(* CODESYS project tc motion control.library
   Author: Adam Garner
   Placeholder: Motion
   Title: Motion
   Version: 0.1.0.0
   Company: Ljmu

Project tree, tasks and I/O mapping:
  libraries: Tc2_MC2, * (Beckhoff Automation GmbH); Tc2_MC2_Drive, * (Beckhoff Automation GmbH); Tc2_Standard, * (Beckhoff Automation GmbH); Tc2_System, * (Beckhoff Automation GmbH); Tc2_Utilities, * (Beckhoff Automation GmbH); Tc3_EventLogger, * (Beckhoff Automation GmbH); Tc3_JsonXml, * (Beckhoff Automation GmbH); Tc3_Module, * (Beckhoff Automation GmbH)
  DUTs/
    data type e_IDXError
    data type e_MCState
    data type e_MotorReadState
    data type ST_IDXError
    data type ST_IDXErrorCode
    data type ST_MCState
  GVLs/
  POUs/
    function block FB_IDXError [ST]: FB_init, GetErrorStructure, IsError, ResetError
    function block FB_IDXReadErrorCode [ST]: ParseErrorCode
    function block FB_IDXReadErrorRegister [ST]: ParseErrorRegister
    function block FB_IDXResetError [ST]
    function block FB_Motion [ST]: Enable, Estop, FB_init, GetAxisRef, GetCurrentPosition, GetStatus, Home, MoveTo, Reset
    function block FB_MotionEventSender [ST]: COEError, EnableMotor, Homing, MotorError, MoveTo, NCReset
    function block FB_ReadErrorStringFromESI [ST]: GetErrorString, StringToUint
    program MAIN [ST]
  VISUs/
*)

// DUTs/e_IDXError
{attribute 'qualified_only'}
{attribute 'strict'}
TYPE e_IDXError :
(
	Generic_Error := 0,
	Current_Error :=1,
	Voltage_Error:=2,
	Temperature_Error:=3,
	Communication_Error := 4,
	Device_Profile_Specific := 5,
	Reserved := 6,
	Motion_Error :=7
);
END_TYPE

// DUTs/e_MCState
{attribute 'qualified_only'}
{attribute 'strict'}
TYPE e_MCState :
(
	Busy,
	Done,
	Error,
	CommandAborted,
	Active,
	Idle
);
END_TYPE

// DUTs/e_MotorReadState
// -27 as is qualified only shouldnt be flagged anyway
{attribute 'strict'}
{attribute 'qualified_only'}
TYPE e_MotorReadState :
(
Idle,
ReadingErrorArray,
{attribute 'analysis' := '-27'}
Parse,
EraseErrorArray,
Waiting,
Error,
CountingErrors,
ReadNextError

);
END_TYPE

// DUTs/ST_IDXError
TYPE ST_IDXError :
STRUCT
	GenericError:BOOL;
	CurrentError : BOOL;
	VoltageError:BOOL;
	TemperatureError:BOOL;
	Communication_Error :BOOL;
	DeviceProfileSpecific :BOOL;
	Reserved :BOOL;
	MotionError :BOOL;
	ErrorCodeArr:ARRAY [0..4] OF ST_IDXErrorCode;


END_STRUCT
END_TYPE

// DUTs/ST_IDXErrorCode
TYPE ST_IDXErrorCode :
STRUCT
	ErrorCode: UINT;
	ErrorString:STRING;
	TimeCode:DT;
END_STRUCT
END_TYPE

// DUTs/ST_MCState
TYPE ST_MCState :
STRUCT
	MCState : e_MCState;
	Done:BOOL;
	CommandAborted:BOOL;
	Status :BOOL;
	Active :BOOL;
	Busy:BOOL;
	Error:BOOL;
	ErrorID:UDINT;
	
END_STRUCT
END_TYPE

// POUs/FB_IDXError
FUNCTION_BLOCK FB_IDXError
// www.maxongroup.com/medias/sys_master/root/8837359632414/IDX-Firmware-Specification-En.pdf 	
VAR
	AxisName 				:STRING;
	ExecuteRead 			: BOOL; 
	MappedErrorCode AT%I* 	: UINT;
	stIDXError 				: ST_IDXError;
	
	fbIDXErrorEventSender 	: FB_MotionEventSender;
	MotorErrorEventSent		: BOOL;


	fbIdxReadErrorCode 		: FB_IDXReadErrorCode;
	NumOfErrorCodes			: USINT;
	ErrorCodeReadError 		: BOOL;
	ErrorCodeAdsErrorCode	: UINT;
	ErrorCodeReadBusy		: BOOL;
	
	fbIDXReadErrorRegister	: FB_IDXReadErrorRegister;
	ErrorRegisterReadError 	: BOOL;
	ErrorRegisterReadBusy	: BOOL;
	ErrorRegisterAdsErrorCode: UINT;
	eErrorRegisterReadState : e_MotorReadState;
	
	fbReadErrorStringFromESI: FB_ReadErrorStringFromESI;
	ErrorStringReadReady 	: BOOL;
	ErrorStringReadBusy 	: BOOL;
	ErrorStringReadError 	: BOOL;
	ErrorStringFound 		: BOOL;
	
	CoeErrorCodeMessageSent : BOOL;
	CoeErrorregisterMessageSent : BOOL;
	
	

	

END_VAR

VAR_INPUT
	Axis 					: AXIS_REF;
END_VAR

VAR_OUTPUT
    Busy         			: BOOL;
    Error        			: BOOL;
END_VAR

VAR CONSTANT
	MaxIndex 				: USINT := 4;
END_VAR

VAR_TEMP
	TempErrorCode 			: UINT;
	TempErrorString 		: STRING;
	Index					: USINT;
END_VAR

// read error Reg 
// check for error messages availible 

IF NOT (MappedErrorCode=0) THEN
	ExecuteRead := TRUE; // motor in error state 
	
ELSE
	ExecuteRead:= FALSE;
END_IF

fbIdxReadErrorCode(
	Axis:= Axis,
	Execute:= ExecuteRead,
	NumOfErrors=> NumOfErrorCodes,
	stErrorInOut:=stIDXError,
	ReadError=>ErrorCodeReadError,
	AdsErrId=>ErrorCodeAdsErrorCode,
	ReadBusy => ErrorCodeReadBusy);

CoeErrorCodeMessageSent := fbIDXErrorEventSender.COEError(
	AxisName := AxisName,
	Error := ErrorCodeReadError,
	AdsErrId:= ErrorCodeAdsErrorCode,
	Description:= 'ErrorCodeRead');

fbIDXReadErrorRegister(
	Axis:= Axis, 
	Execute:= ExecuteRead, 
	stErrorRegisterInOut:=stIDXError , 
	ReadError=> ErrorRegisterReadError, 
	AdsErrId=> ErrorRegisterAdsErrorCode, 
	eMotorReadState=>eErrorRegisterReadState,
	ReadBusy=> ErrorRegisterReadBusy );

CoeErrorregisterMessageSent:= fbIDXErrorEventSender.COEError(
	AxisName:= AxisName,
	Error := ErrorRegisterReadError,
	AdsErrId:= ErrorRegisterAdsErrorCode,
	Description:= 'ErrorCodeRegister');


fbReadErrorStringFromESI(
	ReadyFlag=>ErrorStringReadReady,
	Busy=>ErrorStringReadBusy,
	Error=>ErrorStringReadError);


IF (ErrorStringReadReady AND ExecuteRead ) THEN
	FOR Index:=0  TO MaxIndex BY 1 DO
		TempErrorCode:= stIDXError.ErrorCodeArr[Index].ErrorCode;
		IF NOT (TempErrorCode =0) THEN
			ErrorStringFound:= fbReadErrorStringFromESI.GetErrorString(ErrorCodeIn:= TempErrorCode,ErrorStringOut=>TempErrorString);
			stIDXError.ErrorCodeArr[Index].ErrorString:= TempErrorString;
		END_IF
	END_FOR
END_IF
	
MotorErrorEventSent:= fbIDXErrorEventSender.MotorError(stIDXError:=stIDXError,AxisName:= AxisName);

Busy := ErrorStringReadBusy OR ErrorRegisterReadBusy OR ErrorCodeReadBusy;
Error := ErrorStringReadError OR ErrorRegisterReadError OR ErrorCodeReadError;

METHOD FB_init : BOOL
VAR_INPUT
	bInitRetains : BOOL; // if TRUE, the retain variables are initialized (warm start / cold start)
	bInCopyCode : BOOL;  // if TRUE, the instance afterwards gets moved into the copy code (online change)
	AxisNameIn	:String;
END_VAR
AxisName := AxisNameIn;
END_METHOD

METHOD PUBLIC GetErrorStructure 
VAR_OUTPUT
	StIDXErrorOut : ST_IDXError;
END_VAR
StIDXErrorOut:= stIDXError;
END_METHOD

// returns true if motor is in error state 
METHOD IsError : BOOL
IsError := ExecuteRead;
END_METHOD

METHOD ResetError : BOOL
VAR_IN_OUT
	   		{attribute 'analysis' := '-27'}
	Execute			: BOOL;(*Function block execution is triggered by a rising edge at this input.*)
END_VAR

VAR_INST
	fbCoEWrite		: FB_CoEWrite;
    Data       		: UINT := 16#0080;
    ReadError          	: BOOL;
    AdsErrId       	: UINT;
    CANopenErrId   	: UINT;
END_VAR

VAR CONSTANT
	NetId          	: T_AmsNetID:= '';(*netID of PC with NC*)
   	Index          	: WORD:= 16#6040;(*CoE object index*)
   	SubIndex       	: BYTE:=16#0;(*CoE sub index*)
   	Timeout        	: TIME := DEFAULT_ADS_TIMEOUT;(*States the time before the function is cancelled.*)
  	CompleteAccess 	: BOOL:= FALSE;(*Function block reads the complete object with all sub index*)
END_VAR
IF __ISVALIDREF(Execute) THEN	
	fbCoEWrite(
    NetId          := NetId, 
    Index          := Index, 
    SubIndex       := SubIndex, 
    pSrcBuf        := ADR(Data), 
    BufLen         := USINT_TO_UDINT(SIZEOF(Data)), 
    Execute        := Execute, 
    Timeout        := Timeout, 
    CompleteAccess := CompleteAccess, 
    Axis := Axis
);

END_IF

IF (NOT fbCoEWrite.Busy) AND   __ISVALIDREF(Execute) THEN
    ReadError    := fbCoEWrite.Error;
	IF (NOT ReadError) AND Execute THEN
		ResetError:= TRUE; // reset successfully only shows for one cycle
	ELSE 
		ResetError:= FALSE;
	END_IF
	
    AdsErrId     := fbCoEWrite.AdsErrId;
    CANopenErrId :=fbCoEWrite.CANopenErrId;
    Execute      := FALSE;
	IF NOT ReadError THEN
		ResetError:= TRUE; // reset successfully
	END_IF
END_IF
END_METHOD

END_FUNCTION_BLOCK

// POUs/FB_MotionEventSender
FUNCTION_BLOCK FB_MotionEventSender
VAR
	fbTcMessage : FB_TcMessage;
END_VAR

METHOD COEError : BOOL
VAR_INPUT
    Error        	: BOOL;
    AdsErrId     	: UINT;
	Description		: STRING;
	AxisName		:STRING;
END_VAR
VAR_INST
	LastError		:BOOL;

END_VAR

VAR
	SendResult 			:HRESULT;

	
END_VAR
COEError := FALSE;
IF (NOT LastError) AND Error THEN // only enter is a current error is in place and the last cycle the error was 0 
	 {analysis -9,-46} // Unused  return values and possible use of none init interfaces 
	fbTcMessage.CreateEx(TC_EVENTS.MotionEvents.CoeError,0);
	fbTcMessage.ipArguments.Clear();
	fbTcMessage.ipArguments.AddString(AxisName);
	fbTcMessage.ipArguments.AddUInt(AdsErrId);
	fbTcMessage.ipArguments.AddString(Description);
	SendResult:= fbTcMessage.Send(0);
	{analysis 9,46}
	IF (SendResult=0) THEN
		COEError := TRUE;
	END_IF
END_IF
LastError:= Error;
END_METHOD

METHOD EnableMotor : BOOL
VAR_IN_OUT
	stAxisPowerState : ST_MCState;
END_VAR
VAR_INPUT
	AxisName :STRING;
END_VAR
VAR_INST
	stLastAxisPowerState :ST_MCState;
END_VAR
VAR
	SendResult 			:HRESULT;
	SendEvent :BOOL:= FALSE;
END_VAR
EnableMotor := FALSE;

IF __ISVALIDREF(stAxisPowerState) THEN

	IF NOT (stLastAxisPowerState.MCState = stAxisPowerState.MCState) THEN // state has changed 
	 	{analysis -9,-46} // Unused  return values and possible use of none init interfaces 
		CASE(stAxisPowerState.MCState) OF
		
		e_MCState.Active:
			fbTcMessage.CreateEx(TC_EVENTS.MotionEvents.MotorEnabled,0);
			SendEvent:= TRUE;
		
		e_MCState.Error:
			fbTcMessage.CreateEx(TC_EVENTS.MotionEvents.MotorEnableError,0);
			SendEvent:= TRUE;
		
		e_MCState.Idle:
			fbTcMessage.CreateEx(TC_EVENTS.MotionEvents.MotorDisabled,0);
			SendEvent:= TRUE;
		ELSE
			SendEvent:= FALSE;
		END_CASE
	
		IF SendEvent THEN
			fbTcMessage.ipArguments.Clear();
			fbTcMessage.ipArguments.AddString(AxisName);
			SendResult:= fbTcMessage.Send(0);
			IF (SendResult=0) THEN
				EnableMotor := TRUE;
			END_IF
		END_IF
	END_IF

	stLastAxisPowerState := stAxisPowerState;
END_IF
END_METHOD

METHOD Homing : BOOL
VAR_IN_OUT
	stAxisHomeState : ST_MCState;
END_VAR
VAR_INPUT
	AxisName :STRING;
	ErrorCodeIn :UDINT;
END_VAR
VAR_INST
	stLastAxisHomeState : ST_MCState;
END_VAR
VAR
	SendEvent : BOOL;
	SendResult : Hresult;
END_VAR
Homing := FALSE;

IF  __ISVALIDREF(stAxisHomeState) THEN
	
	IF  (NOT (stLastAxisHomeState.MCState = stAxisHomeState.MCState)) THEN
		CASE(stAxisHomeState.MCState) OF 
		{analysis -9,-46} // Unused  return values and possible use of none init interfaces 
		e_MCState.Done:
			fbTcMessage.CreateEx(TC_EVENTS.MotionEvents.HomeCompleted,0);
			fbTcMessage.ipArguments.Clear();
			fbTcMessage.ipArguments.AddString(AxisName);
			SendEvent := TRUE;
		
		e_MCState.Busy:
			fbTcMessage.CreateEx(TC_EVENTS.MotionEvents.HomeCommandReceived,0);
			fbTcMessage.ipArguments.Clear();
			fbTcMessage.ipArguments.AddString(AxisName);
			SendEvent := TRUE;
		
		e_MCState.Error:
			fbTcMessage.CreateEx(TC_EVENTS.MotionEvents.HomeError,0);
			fbTcMessage.ipArguments.Clear();
			fbTcMessage.ipArguments.AddString(AxisName);
			fbTcMessage.ipArguments.AddUDInt(ErrorCodeIn);
			SendEvent := TRUE;
			
		
		e_MCState.CommandAborted:
			fbTcMessage.CreateEx(TC_EVENTS.MotionEvents.HomeAborted,0);
			fbTcMessage.ipArguments.Clear();
			fbTcMessage.ipArguments.AddString(AxisName);
			SendEvent := TRUE;
			
		e_MCState.Idle:
			SendEvent := FALSE;
		
		ELSE
			SendEvent := FALSE;
			
		
		END_CASE
		
			IF SendEvent THEN
				SendResult:= fbTcMessage.Send(0);
			
				IF (SendResult=0) THEN
					Homing := TRUE;
				END_IF
	
			END_IF
	END_IF
	
	stLastAxisHomeState:= stAxisHomeState;

END_IF
END_METHOD

METHOD PUBLIC MotorError :BOOL
VAR_IN_OUT
	stIDXError 	:ST_IDXError;
END_VAR
VAR_INPUT
	AxisName 	:STRING;
END_VAR
VAR_INST
	stLastIDXError : ST_IDXError;
END_VAR
VAR
	Index :INT;
	ErrorCodeInHex :STRING[255];
	SendResult :HRESULT;
END_VAR
VAR CONSTANT
	MaxIndex :INT := 4 ; 
END_VAR
MotorError:= FALSE;
IF __ISVALIDREF(stIDXError) THEN
FOR Index := 0 TO MaxIndex BY 1 DO 
	IF NOT ( stIDXError.ErrorCodeArr[Index].ErrorCode =stLastIDXError.ErrorCodeArr[Index].ErrorCode) THEN
		{analysis -9,-46,-130}// Unused  return values possible use of none init interfaces ,  Implicit expanding conversion 
		fbTcMessage.CreateEx(TC_EVENTS.MotionEvents.MotorError,0);
		fbTcMessage.ipArguments.Clear();
		fbTcMessage.ipArguments.AddString(AxisName);
		ErrorCodeInHex := DWORD_TO_HEXSTR(stIDXError.ErrorCodeArr[Index].ErrorCode,4,FALSE);
		fbTcMessage.ipArguments.AddString(ErrorCodeInHex);
		fbTcMessage.ipArguments.AddString(stIDXError.ErrorCodeArr[Index].ErrorString);
		SendResult := fbTcMessage.Send(0);
		{analysis 9,46,130}
		IF (SendResult=0) THEN
			MotorError:= TRUE;
		END_IF
		stLastIDXError.ErrorCodeArr[Index]:= stIDXError.ErrorCodeArr[Index];
			
	END_IF
END_FOR
END_IF
END_METHOD

// moveTo bool is true when a event has been sent 
METHOD MoveTo : BOOL
VAR_IN_OUT
	stAxisMoveState : ST_MCState;
END_VAR
VAR_INPUT
	AxisName :STRING;
	TargetPositionIn : LREAL;
	VelocityIn : LREAL;
END_VAR
VAR_INST
	stLastAxisMoveState : ST_MCState;
END_VAR
VAR
	SendEvent : BOOL;
	SendResult : Hresult;
	
END_VAR
MoveTo:= FALSE;
	
IF __ISVALIDREF(stAxisMoveState) THEN
	
	IF  (NOT (stAxisMoveState.MCState = stLastAxisMoveState.MCState)) THEN
	
		CASE(stAxisMoveState.MCState) OF 
		{analysis -9,-46} // Unused  return values and possible use of none init interfaces 	
			e_MCState.Active:
			fbTcMessage.CreateEx(TC_EVENTS.MotionEvents.MotorMoveActive,0);
			fbTcMessage.ipArguments.Clear();
			fbTcMessage.ipArguments.AddString(AxisName);
			SendEvent := TRUE;
	
		e_MCState.Busy:
			fbTcMessage.CreateEx(TC_EVENTS.MotionEvents.MoveCommandReceived,0);
			fbTcMessage.ipArguments.Clear();
			fbTcMessage.ipArguments.AddString(AxisName);
			fbTcMessage.ipArguments.AddLReal(TargetPositionIn);
			fbTcMessage.ipArguments.AddLReal(VelocityIn);
			SendEvent := TRUE;
	
		e_MCState.Error:
			fbTcMessage.CreateEx(TC_EVENTS.MotionEvents.MotorMoveError,0);
			fbTcMessage.ipArguments.Clear();
			fbTcMessage.ipArguments.AddString(AxisName);
			fbTcMessage.ipArguments.AddUDInt(stAxisMoveState.ErrorID);
			SendEvent := TRUE;
	
		e_MCState.CommandAborted:
			fbTcMessage.CreateEx(TC_EVENTS.MotionEvents.MovementAborted,0);
			fbTcMessage.ipArguments.Clear();
			fbTcMessage.ipArguments.AddString(AxisName);
			SendEvent := TRUE;
	
		e_MCState.Done:
			fbTcMessage.CreateEx(TC_EVENTS.MotionEvents.MotorMoveFinshed,0);
			fbTcMessage.ipArguments.Clear();
			fbTcMessage.ipArguments.AddString(AxisName);
			fbTcMessage.ipArguments.AddLReal(TargetPositionIn);
			SendEvent := TRUE;
	
		e_MCState.Idle:
			SendEvent := FALSE;
	
	
		ELSE
			SendEvent := FALSE;
		
		END_CASE
		
		IF SendEvent THEN
			SendResult:= fbTcMessage.Send(0);
			
			IF (SendResult=0) THEN
				MoveTo := TRUE;
			END_IF
		
		END_IF
	
		stLastAxisMoveState := stAxisMoveState;
	
	END_IF

END_IF
END_METHOD

METHOD NCReset : BOOL
VAR_IN_OUT
	stAxisResetState : ST_MCState;
	
END_VAR
VAR_INPUT
	AxisName :STRING;
	ErrorCodeIn :UDINT;
END_VAR
VAR_INST
	stLastAxisResetState : ST_MCState;
END_VAR
VAR
	SendEvent : BOOL;
	SendResult : Hresult;
END_VAR
NCReset := FALSE;

IF  __ISVALIDREF(stAxisResetState) THEN
	
	IF  (NOT (stLastAxisResetState.MCState = stAxisResetState.MCState)) THEN
		CASE(stAxisResetState.MCState) OF 
		{analysis -9,-46} // Unused  return values and possible use of none init interfaces 
		e_MCState.Done:
			fbTcMessage.CreateEx(TC_EVENTS.MotionEvents.NCResetCompleted,0);
			fbTcMessage.ipArguments.Clear();
			fbTcMessage.ipArguments.AddString(AxisName);
			SendEvent := TRUE;
		
		e_MCState.Busy:
			fbTcMessage.CreateEx(TC_EVENTS.MotionEvents.NCResetReceived,0);
			fbTcMessage.ipArguments.Clear();
			fbTcMessage.ipArguments.AddString(AxisName);
			SendEvent := TRUE;
		
		e_MCState.Error:
			fbTcMessage.CreateEx(TC_EVENTS.MotionEvents.NCResetError,0);
			fbTcMessage.ipArguments.Clear();
			fbTcMessage.ipArguments.AddString(AxisName);
			fbTcMessage.ipArguments.AddUDInt(ErrorCodeIn);
			SendEvent := TRUE;
			
		e_MCState.Idle:
			SendEvent := FALSE;
		
		ELSE
			SendEvent := FALSE;
			
		
		END_CASE
		
			IF SendEvent THEN
				SendResult:= fbTcMessage.Send(0);
			
				IF (SendResult=0) THEN
					NCReset := TRUE;
				END_IF
	
			END_IF
	END_IF
	
	stLastAxisResetState:= stAxisResetState;

END_IF
END_METHOD

END_FUNCTION_BLOCK

// POUs/FB_IDXReadErrorCode
// function to read the Diagnosis history odject of a IDX motor 
// this fb will read the errors in the error array looping between them with a 1s pause between reads
// if execute is false it resets the error array no none 
// www.maxongroup.com/medias/sys_master/root/8837359632414/IDX-Firmware-Specification-En.pdf
// definition of motor structure on 6.2.12 pg 71

FUNCTION_BLOCK FB_IDXReadErrorCode
VAR CONSTANT
	 NetId             : T_AmsNetID := ''; // assumes local machine 
    Index             : WORD := 16#10F3; // diagnosis history 
    Timeout           : TIME := T#5S;
    CompleteAccess    : BOOL := FALSE; // to read the whole index in one go instead of sunindexs
	NumberOfErrors :USINT := 5; // number of errors 
	MaxErrorIndex :USINT := 4; // max index so one below number of errors 
	MotorErrorSubindexStart :USINT := 6 ;

END_VAR

VAR_INPUT
	Axis :AXIS_REF;// used For Coe read 
		 {attribute 'analysis' := '-27'}
	Execute: BOOL;	
END_VAR
VAR_IN_OUT
	stErrorInOut : ST_IDXError;// a array for errors with code string and datetime 
END_VAR
VAR_OUTPUT
	NumOfErrors :USINT; // how man errors are present 
	ReadError :BOOL; // error reading motor 
	AdsErrId  : UINT; //holds Reading error codes 
	ReadBusy:BOOL;
END_VAR

VAR
	eMotorReadState : e_MotorReadState; // enum of fb  current state
	
	CoETimer : TON:= (PT:= T#1S); // timer 
	TimerStart:BOOL:= FALSE;
	TimerElapsed:BOOL;
	fbCoERead         : FB_CoERead; // fb to Coe read
    SubIndex          : BYTE := 16#6;  // first error index 
    ExecuteRead       : BOOL := FALSE;
    Error             : BOOL;
    CANopenErrId      : UINT; 
	ParsingError	: BOOL;
	
	ParsedErrorCode : ST_IDXErrorCode;
	ErrorIndex :BYTE := 0; // where to save the error code in the error array 
	RawErrorArray :ARRAY[0..15] OF USINT; // buffer to store the raw CoE Read
	EmptyError : ST_IDXError; // used to reinitalise the error array while not in error state 
END_VAR
VAR_TEMP
		ArrayIndex:USINT;
END_VAR


fbCoERead(
    NetId          := NetId, 
    Index          := Index, 
    SubIndex       := SubIndex, 
    pDstBuf        := ADR(RawErrorArray), 
    BufLen         := USINT_TO_UDINT(SIZEOF(RawErrorArray)), 
    Execute        := ExecuteRead, 
    Timeout        := Timeout, 
    CompleteAccess := CompleteAccess, 
    Axis           := Axis,
	Busy			=> ReadBusy 
); // read the Coe 



CoETimer(IN:= TimerStart,Q=>TimerElapsed); // process timer

CASE(eMotorReadState) OF 
	
e_MotorReadState.Idle: // not reading
	//reset counters
	SubIndex := MotorErrorSubindexStart ;// first error in  motor error array
	ErrorIndex := 0; // first error in output array
	NumOfErrors:= 0;
	
	IF Execute THEN
		ExecuteRead := TRUE;
		eMotorReadState := e_MotorReadState.ReadingErrorArray;
	ELSE 
		IF __ISVALIDREF(stErrorInOut) THEN
			stErrorInOut:= EmptyError; 
		 END_IF
		 
	
		
	END_IF

e_MotorReadState.ReadingErrorArray:

IF NOT (fbCoERead.Busy) THEN // finished reading so write any errors to varibles 
	Error        :=fbCoERead.Error; 
    AdsErrId     :=fbCoERead.AdsErrId;
    CANopenErrId :=fbCoERead.CANopenErrId;
    ExecuteRead  := FALSE; // Reset Reading FB
    
	ReadError:= Error; // if a read fails put into error state 
	ParseErrorCode(ErrorArrayIn:= RawErrorArray,ParsedErrorOut=> ParsedErrorCode,Error=> ParsingError);
	
	IF NOT ParsingError OR Error THEN // if errored dont write to array 
	stErrorInOut.ErrorCodeArr[ErrorIndex]:= ParsedErrorCode;
	END_IF
	
	IF (ErrorIndex = MaxErrorIndex) THEN //  has read whole array 
		eMotorReadState := e_MotorReadState.CountingErrors; //Count and then waiting timer
	ELSE
		eMotorReadState:= e_MotorReadState.ReadNextError;
	END_IF
	

	
	
END_IF

e_MotorReadState.ReadNextError:

ErrorIndex := (ErrorIndex+1) MOD NumberOfErrors; // loop from the error indexs 0 to 4 
SubIndex := ErrorIndex + MotorErrorSubindexStart; // Subindex to read from the motor subindexs 6 to 10 contain errors 
ExecuteRead:= TRUE;
eMotorReadState:= e_MotorReadState.ReadingErrorArray;

e_MotorReadState.CountingErrors:
NumOfErrors := 0;
IF __ISVALIDREF(stErrorInOut) THEN
	FOR ArrayIndex := 0 TO MaxErrorIndex BY 1 DO 
		IF NOT (stErrorInOut.ErrorCodeArr[ArrayIndex].ErrorCode =0) THEN 
		 {analysis -38}
			NumOfErrors := (NumOfErrors +1);
		END_IF
	END_FOR
END_IF
eMotorReadState := e_MotorReadState.Waiting;

e_MotorReadState.Waiting:
TimerStart:= TRUE; // start waiting timer 
IF TimerElapsed THEN
	TimerStart:= FALSE; // reset timer 
	eMotorReadState := e_MotorReadState.Idle; // back to begining 
END_IF

e_MotorReadState.Parse:
// no code needed
e_MotorReadState.EraseErrorArray:
// no code needed

e_MotorReadState.Error:
SubIndex := 6 ;// first error in  motor error array
ErrorIndex := 0; // first error in output array
// Erase error array as not currently reading error 
NumOfErrors:= 0;
ExecuteRead := FALSE;
eMotorReadState := e_MotorReadState.Idle;		



ELSE 
	eMotorReadState := e_MotorReadState.Idle;

END_CASE



// example packet for error 8A81
//00 E0 81 8A 02 00 81 8A 00 00 00 00 00 00 00 00
//0  1  2  3  4  5  6  7  8  9  10 11 12 13 14 15

METHOD ParseErrorCode  
VAR_IN_OUT
ErrorArrayIn :ARRAY[0..15] OF USINT;
END_VAR

VAR_OUTPUT
	ParsedErrorOut : ST_IDXErrorCode;
	Error:BOOL;
END_VAR

VAR
	RawErrorCodes : ARRAY [0..1] OF UINT;
	FirstErrorByte : UINT;
	SecondErrorByte : UINT;
	
END_VAR

VAR CONSTANT
	BlankArray : ARRAY[0..15] OF USINT := [0,0,0,0,0,0,0,0,0,0,0,0,0,0,0,0] ;
END_VAR
Error:= FALSE;
IF __ISVALIDREF(ErrorArrayIn) THEN
	// grab from the first time the error is wrote packets 3&4
	FirstErrorByte := SHL(USINT_TO_UINT(ErrorArrayIn[3]),8);// grab first byte and shift left 
	SecondErrorByte := USINT_TO_UINT(ErrorArrayIn[2]);  // grab second byte 
	RawErrorCodes[0] := FirstErrorByte OR SecondErrorByte; // combine 

	// grab from the Second time the error is wrote packets 6&7
	FirstErrorByte := SHL(USINT_TO_UINT(ErrorArrayIn[7]),8);// grab first byte and shift left 
	SecondErrorByte := USINT_TO_UINT(ErrorArrayIn[6]);  // grab second byte 
	RawErrorCodes[1] := FirstErrorByte OR SecondErrorByte; // combine 
ELSE 
	Error:= TRUE;
END_IF

IF NOT RawErrorCodes[0] = RawErrorCodes[1] THEN
	Error:= TRUE;
ELSE
	ParsedErrorOut.ErrorCode:= RawErrorCodes[0]; 

	


END_IF
// clear array after parsing 
ErrorArrayIn := BlankArray;
END_METHOD

END_FUNCTION_BLOCK

// POUs/FB_IDXReadErrorRegister
FUNCTION_BLOCK FB_IDXReadErrorRegister
VAR_INPUT
	Axis :Axis_Ref;// used For Coe read 
	Execute: BOOL;	
END_VAR
VAR_IN_OUT
	stErrorRegisterInOut :  ST_IDXError;// a array for errors with code string and datetime 
END_VAR
VAR_OUTPUT
	ReadError :BOOL; // error reading motor 
	AdsErrId  : UINT; //holds Reading error codes 
	eMotorReadState : e_MotorReadState; // enum of fb  current state
	ReadBusy :BOOL;
END_VAR

VAR

	CoETimer : TON:= (PT:= T#1S); // timer 
	TimerStart:BOOL:= FALSE;
	TimerElapsed:BOOL;
	fbCoERead         : FB_CoERead; // fb to Coe read
    NetId             : T_AmsNetID := ''; // assumes local machine 
    Index             : WORD := 16#1001; // diagnosis history 
    SubIndex          : BYTE := 16#0;  // first error index 
    ExecuteRead       : BOOL := FALSE;
    Timeout           : TIME := T#5S;
    CompleteAccess    : BOOL := FALSE; // to read the whole index in one go instead of sunindexs
    Error             : BOOL;
    CANopenErrId      : UDINT;
	ParsingError	: BOOL;
	ParsedErrorRegister : ST_IDXErrorCode;
	RawErrorRegister : USINT; // buffer to store the raw CoE Read
	EmptyError : ST_IDXError; // used to reinitalise the error array while not in error state
END_VAR

fbCoERead(
    NetId          := NetId, 
    Index          := Index, 
    SubIndex       := SubIndex, 
    pDstBuf        := ADR(RawErrorRegister), 
    BufLen         := SIZEOF(RawErrorRegister), 
    Execute        := ExecuteRead, 
    Timeout        := Timeout, 
    CompleteAccess := CompleteAccess, 
    Axis           := Axis,
	Busy			=> ReadBusy 
); // read the Coe 



CoETimer(IN:= TimerStart,Q=>TimerElapsed); // process timer

CASE(eMotorReadState) OF 
	
e_MotorReadState.Idle: // not reading
	IF Execute THEN
	ExecuteRead := TRUE;
	eMotorReadState := e_MotorReadState.ReadingErrorArray;
	ELSE // Erase error array as not currently reading error 
		stErrorRegisterInOut:= EmptyError;
	END_IF

e_MotorReadState.ReadingErrorArray:
IF NOT ReadBusy THEN // finished reading so write any errors to varibles 
	Error        :=fbCoERead.Error; 
    AdsErrId     :=fbCoERead.AdsErrId;
    CANopenErrId :=fbCoERead.CANopenErrId;
    ExecuteRead      := FALSE; // Reset Reading FB as finished reading
	ReadError:= Error; // if a read fails Flag Error
	IF NOT ReadError THEN// add data to structure
		ParseErrorRegister(ErrorRegIn:= RawErrorRegister,StErrorRegister:= stErrorRegisterInOut); 
	END_IF
	eMotorReadState := e_MotorReadState.Waiting; // start the waiting timer 
END_IF

e_MotorReadState.Waiting:
TimerStart:= TRUE; // start waiting timer 
IF TimerElapsed THEN
	TimerStart:= FALSE; // reset timer 
	eMotorReadState := e_MotorReadState.Idle; // back to begining 
END_IF

	
END_CASE

METHOD ParseErrorRegister : BOOL
VAR_INPUT
	ErrorRegIn :USINT;
END_VAR
VAR_IN_OUT
	StErrorRegister :ST_IDXError;
END_VAR
StErrorRegister.GenericError := ErrorRegIn.0;
StErrorRegister.CurrentError := ErrorRegIn.1;
StErrorRegister.VoltageError := ErrorRegIn.2;
 StErrorRegister.TemperatureError := ErrorRegIn.3;
StErrorRegister.Communication_Error := ErrorRegIn.4;
StErrorRegister.DeviceProfileSpecific := ErrorRegIn.5;
StErrorRegister.MotionError := ErrorRegIn.7;
END_METHOD

END_FUNCTION_BLOCK

// POUs/FB_ReadErrorStringFromESI
// functionblock async creates error codes from the maxons IDX ESI file 
// the ESI structure is below except with more error codes 

//<EtherCATInfo Version="1.2" xmlns:xsi="http://www.w3.org/2001/XMLSchema-instance" xsi:noNamespaceSchemaLocation="EtherCATInfo.xsd">
// 	<Descriptions>
//		<Devices>
//			<Device Physics="YY">
//				<Profile>
//					<DiagMessages>
//						<DiagMessage>
//             				<TextId>#x0000</TextId>
//             				<MessageText>None</MessageText>
//           			</DiagMessage>
//           			<DiagMessage>
//            				<TextId>#x1000</TextId>
//            				<MessageText>Generic error</MessageText>
//          			</DiagMessage>
//					<DiagMessages>
//				</Profile>
//			</Device Physics="YY">
//		</Devices>
// 	</Descriptions>
//</EtherCATInfo Version="1.2" xmlns:xsi="http://www.w3.org/2001/XMLSchema-instance" xsi:noNamespaceSchemaLocation="EtherCATInfo.xsd">


FUNCTION_BLOCK FB_ReadErrorStringFromESI
VAR_OUTPUT
	Busy:BOOL;
	Error :BOOL;
	ReadyFlag :BOOL; 
END_VAR
VAR
	{attribute 'strict'}
	eXMLReadState : (LoadingFile,GettingIterator,ParsingFile,Ready,ErrorState);
 	{attribute 'analysis' := '-26'} // string truncated to 80 char
	ErrorCodeStringArray : ARRAY [0..16#FFFF] OF STRING;
	fbXml : FB_XmlDomParser; // init fb 
	LoadFile:BOOL:= TRUE; 
	FileLoaded:BOOL; // latches true once file opened
	xmlDoc: SXmlNode; // root node
	xmlEtherCatInfo :SXmlNode; // <ethercatInfo> Node
	xmlDescriptions :SXmlNode;// <Descriptions> Node 
	xmlDevices : SXmlNode; // <Devices> Node 
	xmlDevice : SXmlNode;// <Device Physics="YY"> Node 
	xmlProfile : SXmlNode;//<Profile> Node
	xmlDiagMessages:SxmlNode;// <DiagMessages> Node
	xmlDiagmessageIterator:SXmlIterator;//<DiagMessage> iterator
	xmlDiagMessage :SXmlNode; // individual <DiagMessage> nodes
	xmlDiagMessageIDNode :sxmlNode; // individual <TextId> node
	xmlDiagMessageMessageTextNode : SxmlNode;// individual <MessageText> node

	xmlDiagMessageIDText:STRING[255];
	ErrorCode :UINT;
	StringToUintError :BOOL;
	

	DiagMessageIteratorLoaded :BOOL := FALSE;




END_VAR
VAR CONSTANT
	NumToItetratePerCycle :UINT := 25; // controls number of messages read in a cycle 
END_VAR
VAR_TEMP
	
	ErrorString: STRING[80];
	DiagMessageIndex : UINT ; 
END_VAR

CASE eXMLReadState OF 
	LoadingFile :
		
		Busy:=TRUE;
		IF LoadFile THEN
		FileLoaded:= fbXml.LoadDocumentFromFile(
		sFile:= 'C:\TwinCAT\3.1\Config\Io\EtherCAT\maxon_motor_IDX_0170h_6650h_0000h_0000h_ESI.xml',
		bExec:= LoadFile,
		);
		ELSE
			eXMLReadState := GettingIterator;
		END_IF

	
	GettingIterator : 
	IF NOT FileLoaded THEN
		eXMLReadState := ErrorState;
	END_IF
		Busy:= FALSE;
		DiagMessageIteratorLoaded:=TRUE;
		xmlDoc:= fbXml.GetDocumentNode();
		xmlEtherCatInfo := fbXml.ChildByName(xmlDoc, 'EtherCATInfo');
		xmlDescriptions := fbXml.ChildByName(xmlEtherCatInfo, 'Descriptions');
		xmlDevices := fbXml.ChildByName(xmlDescriptions, 'Devices');
		xmlDevice := fbXml.ChildByAttributeAndName(xmlDevices, 'Physics', 'YY', 'Device');
		xmlProfile := fbXml.ChildByName(xmlDevice, 'Profile');
		xmlDiagMessages := fbXml.ChildByName(xmlProfile, 'DiagMessages');
		xmlDiagmessageIterator:= fbXml.Begin(xmlDiagMessages);
		eXMLReadState := ParsingFile;
	
	ParsingFile : 
			FOR DiagMessageIndex:=0  TO NumToItetratePerCycle BY 1 DO // loop 0 to 25 
		IF NOT fbXml.IsEnd(xmlDiagmessageIterator) THEN// Still messages to Parse 
			xmlDiagMessage := fbXml.Node(xmlDiagmessageIterator); //  <DiagMessage> node
  			xmlDiagMessageIDNode :=  fbXml.ChildByName(xmlDiagMessage, 'TextId');// find the <TextID> in the level below 
  			xmlDiagMessageIDText := fbXml.NodeText(xmlDiagMessageIDNode);// pull out the text 
			StringToUintError:= StringToUint(ErrorCodeString := xmlDiagMessageIDText ,ErrorCodeOut=> ErrorCode);
			xmlDiagMessageMessageTextNode :=  fbXml.ChildByName(xmlDiagMessage, 'MessageText');// find the <MessageText> 
			 {analysis -26}
	  		ErrorString := fbXml.NodeText(xmlDiagMessageMessageTextNode);// pull out the text 
			 
			ErrorCodeStringArray[ErrorCode] := ErrorString;
			xmlDiagmessageIterator := fbXml.Next(xmlDiagmessageIterator);
		ELSE
			eXMLReadState := Ready;	
		END_IF
		
		END_FOR
	
	Ready :
		ReadyFlag:= TRUE;
	ErrorState:
		Error:=TRUE;
		
	
	ELSE // in case a undefined Enum
		eXMLReadState := LoadingFile;
END_CASE

// returns true if a String is found for that error code 
METHOD GetErrorString : BOOL
VAR_INPUT
		ErrorCodeIn:UINT;
END_VAR
VAR_OUTPUT
   		{attribute 'analysis' := '-23'}
		ErrorStringOut:STRING;
END_VAR
IF (ErrorCodeStringArray[ErrorCodeIn] = '')THEN
	GetErrorString := FALSE; 
ELSE
	GetErrorString := TRUE; 
END_IF


ErrorStringOut := ErrorCodeStringArray[ErrorCodeIn];
END_METHOD

// input string example '#xFFFF'
METHOD PUBLIC StringToUint :BOOL
VAR_INPUT
	ErrorCodeString :STRING[8];
END_VAR
VAR_OUTPUT 
	ErrorCodeOut :UINT;
END_VAR
VAR
	DataOutput : ARRAY[0..1] OF BYTE;
	FormattedString :STRING[255];
	SpacedString : STRING[255];
	ErrorCodeTemp :UINT;
	BytesWrote:UDINT;
END_VAR
FormattedString := RIGHT (STR:= ErrorCodeString,SIZE:= 4); // removes'#x'
SpacedString := INSERT(STR1:= FormattedString,STR2:=' ', POS := 2); // inserts a space between bytes 
BytesWrote:= HEXSTR_TO_DATA(sHex := SpacedString,pData:= ADR(DataOutput),cbData:= USINT_TO_UDINT(SIZEOF(DataOutput)));// Function Wants 'AB CD'
ErrorCodeTemp := SHL(BYTE_TO_UINT(DataOutput[0]),8);
ErrorCodeTemp := ErrorCodeTemp OR BYTE_TO_UINT(DataOutput[1]);
IF NOT (BytesWrote=2) THEN 
	StringToUint:=FALSE;
ELSE
	ErrorCodeOut := ErrorCodeTemp;
	StringToUint:=TRUE;
END_IF
END_METHOD

END_FUNCTION_BLOCK

// POUs/FB_IDXResetError
FUNCTION_BLOCK FB_IDXResetError 
VAR_IN_OUT
	Execute			: BOOL;(*Function block execution is triggered by a rising edge at this input.*)
END_VAR

VAR_INPUT
	Axis			: AXIS_REF;
END_VAR
VAR
	fbCoEWrite		: FB_CoEWrite;
    Data       		: UINT := 16#0080;
    Error          	: BOOL;
    AdsErrId       	: UINT;
    CANopenErrId   	: UINT;
END_VAR
VAR CONSTANT
	NetId          	: T_AmsNetID:= '';(*netID of PC with NC*)
   	Index          	: WORD:= 16#6040;(*CoE object index*)
   	SubIndex       	: BYTE:=16#0;(*CoE sub index*)
   	Timeout        	: TIME := DEFAULT_ADS_TIMEOUT;(*States the time before the function is cancelled.*)
  	CompleteAccess 	: BOOL:= FALSE;(*Function block reads the complete object with all sub index*)
END_VAR


IF __ISVALIDREF(Execute) THEN	
	fbCoEWrite(
    NetId          := NetId, 
    Index          := Index, 
    SubIndex       := SubIndex, 
    pSrcBuf        := ADR(Data), 
    BufLen         := USINT_TO_UDINT(SIZEOF(Data)), 
    Execute        := Execute, 
    Timeout        := Timeout, 
    CompleteAccess := CompleteAccess, 
    Axis := Axis
);

END_IF

IF (NOT fbCoEWrite.Busy AND   __ISVALIDREF(Execute)) THEN
    Error        := fbCoEWrite.Error;
    AdsErrId     := fbCoEWrite.AdsErrId;
    CANopenErrId :=fbCoEWrite.CANopenErrId;
    Execute      := FALSE;
END_IF

END_FUNCTION_BLOCK

// POUs/FB_Motion
FUNCTION_BLOCK FB_Motion
VAR_INPUT
END_VAR
VAR_OUTPUT
END_VAR
VAR
	Axis: AXIS_REF;
	AxisName :STRING;
	fbMotionEventSender : FB_MotionEventSender;
	
	
	fbAxisPower: MC_Power;
	stAxisPowerState : ST_MCState;
	
	fbAxisHalt : MC_Halt;
	stAxisHaltState : ST_MCState;
	
	fbAxisMove : MC_MoveAbsolute;
	stAxisMoveState : ST_MCState;
	
	fbAxisReset : MC_Reset;
	stAxisResetState :ST_MCState;
	
	fbAxisHome : MC_Home;
	stAxisHomeState : ST_MCState;
END_VAR

Axis.ReadStatus();

METHOD PUBLIC Enable : BOOL
VAR_INPUT
	Execute :BOOL;
END_VAR
VAR
	EventSent :bool;
END_VAR
fbAxisPower( // use in idx class
    Axis:= Axis,
    Enable:= Execute,
    Enable_Positive:= Execute,
    Enable_Negative:= Execute,
	BufferMode := MC_Aborting,
    Override:= 100.0,
	Status=>stAxisPowerState.Status,
	Error=>stAxisPowerState.Error,
	ErrorID => stAxisPowerState.ErrorID,
	Busy => stAxisPowerState.Busy
);

IF stAxisPowerState.Status THEN // axis is enabled
	stAxisPowerState.MCState := e_MCState.Active;
	
ELSIF stAxisPowerState.Busy THEN // fb is busy while enabling or axis is enabled
	stAxisPowerState.MCState := e_MCState.Busy;
	
ELSIF stAxisPowerState.Error THEN // in error state 
	stAxisPowerState.MCState := e_MCState.Error;
ELSE 
	stAxisPowerState.MCState := e_MCState.Idle;
END_IF


EventSent:= fbMotionEventSender.EnableMotor(
	stAxisPowerState:= stAxisPowerState,
	AxisName:= AxisName);
END_METHOD

METHOD Estop : BOOL
VAR_INPUT
	Execute :bool;
END_VAR
fbAxisHalt(
	Axis:=Axis, 
	Execute:= Execute, 
	Deceleration:= , 
	Jerk:= , 
	BufferMode:=MC_Aborting ,  
	Done=> stAxisHaltState.Done, 
	Busy=>stAxisHaltState.Busy , 
	Active=>stAxisHaltState.Active , 
	CommandAborted=>stAxisHaltState.CommandAborted , 
	Error=>stAxisHaltState.Error , 
	ErrorID=> stAxisHaltState.ErrorID );
	
	

IF stAxisHaltState.Done THEN // axis been stopped 
		stAxisHaltState.MCState:= e_MCState.Done;
		
	ELSIF stAxisHaltState.Busy THEN 
		stAxisHaltState.MCState:= e_MCState.Busy;
		
	ELSIF stAxisHaltState.Error THEN	
		stAxisHaltState.MCState:= e_MCState.Error;
		
	ELSIF stAxisHaltState.CommandAborted THEN	
		stAxisHaltState.MCState:= e_MCState.CommandAborted;
		
	ELSE
		stAxisHaltState.MCState:= e_MCState.Idle;

	
END_IF
END_METHOD

METHOD FB_init : BOOL
VAR_INPUT
	bInitRetains : BOOL; // if TRUE, the retain variables are initialized (warm start / cold start)
	bInCopyCode : BOOL;  // if TRUE, the instance afterwards gets moved into the copy code (online change)
	AxisNameIn :string;
END_VAR
AxisName := AxisNameIn;
END_METHOD

METHOD PUBLIC GetAxisRef
VAR_OUTPUT
	AxisRefOut : AXIS_REF;
END_VAR
AxisRefOut := Axis;
END_METHOD

METHOD PUBLIC GetCurrentPosition
VAR_OUTPUT
	PositionOut :LREAL;
END_VAR
PositionOut:= Axis.NcToPlc.ActPos;
END_METHOD

METHOD GetStatus : BOOL
VAR_OUTPUT
	AxisOut :ST_AxisStatus;
END_VAR
AxisOut := Axis.Status;
END_METHOD

METHOD PUBLIC Home : BOOL
VAR_IN_OUT
	Execute :BOOL;
END_VAR

VAR_INPUT
		HomePositionIn :LREAL;
END_VAR
	fbAxisHome(
	Axis:=Axis,
	Execute:=Execute,
	Position:=HomePositionIn,
	HomingMode:=MC_DefaultHoming,
	Busy=>stAxisHomeState.Busy,
	Done=>stAxisHomeState.Done,
	Error=> stAxisHomeState.Error,
	ErrorID=> stAxisHomeState.ErrorID);

	
	IF stAxisHomeState.Done THEN // axis been Homed 
		stAxisHomeState.MCState:= e_MCState.Done;
		
	ELSIF stAxisHomeState.Busy THEN // 
		stAxisHomeState.MCState:= e_MCState.Busy;
		
	ELSIF stAxisHomeState.Error THEN	
		stAxisHomeState.MCState:= e_MCState.Error;
		
	ELSIF stAxisHomeState.CommandAborted THEN	
		stAxisHomeState.MCState:= e_MCState.CommandAborted;
		
	ELSE
		stAxisHomeState.MCState:= e_MCState.Idle;

END_IF

IF stAxisHomeState.Busy THEN
	Execute := FALSE;
END_IF
 Home:= stAxisHomeState.Busy;
 
 fbMotionEventSender.Homing(
	stAxisHomeState:= stAxisHomeState,
	AxisName:= AxisName,
	ErrorCodeIn:= stAxisHomeState.ErrorID);
END_METHOD

METHOD PUBLIC MoveTo : BOOL
VAR_INPUT
	TargetPositionIn : LREAL;
	VelocityIn : LREAL;
END_VAR

VAR_IN_OUT
		Execute :BOOL;
END_VAR
VAR_OUTPUT
	eStateOut : e_MCState;
END_VAR
VAR
	EventSent	: bool;
END_VAR
fbAxisMove(
	Axis:= Axis, 
	Execute:= Execute, 
	Position:= TargetPositionIn, 
	Velocity:= VelocityIn, 
	BufferMode:= MC_BufferMode.MC_BlendingNext , 
	Done=>stAxisMoveState.Done , 
	Busy=> stAxisMoveState.Busy, 
	Active=> stAxisMoveState.Active, 
	CommandAborted=> stAxisMoveState.CommandAborted, 
	Error=>stAxisMoveState.Error , 
	ErrorID=> stAxisMoveState.ErrorID);
	
IF stAxisMoveState.Active THEN // axis In Motion
		stAxisMoveState.MCState:= e_MCState.Active;
		
	ELSIF stAxisMoveState.Busy THEN // fb busy
		stAxisMoveState.MCState:= e_MCState.Busy;
		
	ELSIF stAxisMoveState.Error THEN	
		stAxisMoveState.MCState:= e_MCState.Error;
		
	ELSIF stAxisMoveState.CommandAborted THEN	
		stAxisMoveState.MCState:= e_MCState.CommandAborted;
		
	ELSIF stAxisMoveState.Done THEN
		stAxisMoveState.MCState := e_MCState.Done;
		
	ELSE
		stAxisMoveState.MCState:= e_MCState.Idle;

END_IF

eStateOut:= stAxisMoveState.MCState;

IF stAxisMoveState.Busy THEN
	Execute := FALSE;
END_IF


EventSent:= fbMotionEventSender.MoveTo(
	stAxisMoveState:= stAxisMoveState,
	AxisName:= AxisName,
	TargetPositionIn:= TargetPositionIn,
	VelocityIn:= VelocityIn);
END_METHOD

METHOD PUBLIC Reset : BOOL
VAR_INPUT
	Execute:bool;
END_VAR

VAR

END_VAR
Reset := FALSE;
fbAxisReset(
	Axis:= Axis , 
	Execute:= Execute, 
	Done=> stAxisResetState.Done, 
	Busy=> stAxisResetState.Busy, 
	Error=>stAxisResetState.Error , 
	ErrorID=>stAxisResetState.ErrorID);
	
IF stAxisResetState.Done THEN
	stAxisResetState.MCState := e_MCState.Done;
		
	ELSIF stAxisResetState.Busy THEN
		stAxisResetState.MCState := e_MCState.Busy;
END_IF

IF stAxisResetState.Error THEN
	stAxisResetState.MCState:= e_MCState.Error;
END_IF

fbMotionEventSender.NCReset(
	stAxisResetState:= stAxisResetState,
	AxisName:= AxisName,
	ErrorCodeIn:= stAxisResetState.ErrorID);
END_METHOD

END_FUNCTION_BLOCK

// POUs/MAIN
{attribute 'analysis' := '-33,-2'}
PROGRAM MAIN
VAR

	fbReadErrorCodeFromESI : FB_ReadErrorStringFromESI;
END_VAR

END_PROGRAM
